// TwinCAT 3 PLC project SPS_Main_Proj
// ProgramVersion: 3.1.4024.0
// libraries:
//   Tc2_Standard, * (Beckhoff Automation GmbH)
//   Tc2_System, * (Beckhoff Automation GmbH)
//   Tc3_Module, * (Beckhoff Automation GmbH)
// project tree:
//   GVLs/ GVL_Liste1.TcGVL
//   / PlcTask.TcTTO
//   POUs/ F_AdditionFunction.TcPOU, F_SubstractFunction.TcPOU, F_MultiplicationFunction.TcPOU, F_DivisionFunction.TcPOU, MAIN.TcPOU, PRG_DoSomeMath.TcPOU
// real-time tasks:
//   TASK PlcTask: cycle T#10ms, priority 20, ADS port 350

CONFIGURATION SPS_Main_Proj
    RESOURCE PLC ON TwinCAT3
        TASK PlcTask(INTERVAL := T#10ms, PRIORITY := 20);
        PROGRAM MAIN WITH PlcTask : MAIN;
    END_RESOURCE
END_CONFIGURATION

// ---- GVLs/GVL_Liste1.TcGVL
{attribute 'qualified_only'}
VAR_GLOBAL
	rEps : REAL := 1E-9;
	
END_VAR

// ---- POUs/MAIN.TcPOU
PROGRAM MAIN
VAR
	bTasterBlau 	: BOOL := TRUE; //bool
	uiZaehlerObjekt	: UINT := 23; //uint 16bit
	rTemp			: REAL := -3.34; //float 16bit
	(*
	Kommentar
	*)
	rAdditionResult : REAL;
END_VAR

IF bTasterBlau THEN
	uiZaehlerObjekt := uiZaehlerObjekt +1;
END_IF

rAdditionResult := F_AdditionFunction(4.3,3.4);

PRG_DoSomeMath();

END_PROGRAM

// ---- POUs/F_AdditionFunction.TcPOU
FUNCTION F_AdditionFunction : REAL
VAR_INPUT
	rInput1 : REAL;
	rInput2 : REAL;
END_VAR
VAR
END_VAR

F_AdditionFunction := rInput1 + rInput2;

END_FUNCTION

// ---- POUs/PRG_DoSomeMath.TcPOU
PROGRAM PRG_DoSomeMath
VAR_INPUT
	
END_VAR
VAR
	rVariable1 : REAL;
	rVariable2 : REAL;
	rVariable3 : REAL;
	rVariable4 : REAL;
	rPRG_Count : UINT;
END_VAR

rPRG_Count := rPRG_Count + 1;

rVariable1 := F_AdditionFunction(23.23,4.3);
rVariable2 := F_SubstractFunction(23.23,4.3);
rVariable3 := F_MultiplicationFunction(23.23,4.3);
rVariable4 := F_DivisionFunction(23.23,4.3);

END_PROGRAM

// ---- POUs/F_SubstractFunction.TcPOU
FUNCTION F_SubstractFunction : REAL
VAR_INPUT
	rInput1 : REAL;
	rInput2 : REAL;
END_VAR
VAR
END_VAR

F_SubstractFunction := rInput1 - rInput2;

END_FUNCTION

// ---- POUs/F_MultiplicationFunction.TcPOU
FUNCTION F_MultiplicationFunction : REAL
VAR_INPUT
	rInput1 : REAL;
	rInput2 : REAL;
END_VAR
VAR
END_VAR

F_MultiplicationFunction := rInput1 * rInput2;

END_FUNCTION

// ---- POUs/F_DivisionFunction.TcPOU
FUNCTION F_DivisionFunction : REAL
VAR_INPUT
	rInput1 : REAL;
	rInput2 : REAL;
END_VAR
VAR
END_VAR

IF rInput2 < GVL_Liste1.rEps THEN
	F_DivisionFunction := 0;
ELSE
	F_DivisionFunction := rInput1 / rInput2;
END_IF

END_FUNCTION
